// TIA Portal V17 export
// export: Created 2025-03-11T12:28:50.280284Z, ExportSetting WithDefaults, DisplayName Totally Integrated Automation Portal, DisplayVersion V17 Update 8, DisplayName TIA Portal Openness, DisplayVersion V17 Update 8, DisplayName TIA Portal Version Control Interface, DisplayVersion V17, DisplayName SINAMICS Startdrive Advanced, DisplayVersion V17 SP2, DisplayName SINAMICS Startdrive G110M, G120, G120C, G120D, G120P, G115D, DisplayVersion V17 SP2, DisplayName SINAMICS Startdrive G130, G150, S120, S150, SINAMICS MV, S210, DisplayVersion V17 SP2, DisplayName STEP 7 Professional, DisplayVersion V17 Update 8, DisplayName SINUMERIK ONE STEP 7 Toolbox, DisplayVersion V17 Update 12, DisplayName SINUMERIK 840D sl STEP 7 Toolbox, DisplayVersion V17 Update 12, DisplayName STEP 7 Safety, DisplayVersion V17 Update 6, DisplayName WinCC Advanced, DisplayVersion V17 Update 8
FUNCTION_BLOCK "FB21222_POWDER_FILLING_START_STOP_BY_CURRENT"   // FB21222, LAD
{ S7_Optimized_Access := 'TRUE' }
VERSION : 0.1
// stored: AutoNumber false, IsIECCheckEnabled false, IsRetainMemResEnabled false, MemoryReserve 100, SetENOAutomatically false, UDAEnableTagReadback false
   VAR_INPUT
      SENSOR_VALUE : Int;   // SENSOR VALUE
      iFEEDER_STATE_LINE : Word;
      HMI_HIGH_CURRENT_LIMIT : Real;   // HMI HIGH CURRENT LIMIT
      HMI_LOW_CURRENT_LIMIT : Real;   // HMI LOW CURRENT LIMIT
   END_VAR
   VAR_OUTPUT
      POWDER_FILLING_STOP_BY_CURRENT : Bool;   // HMI POWDER FILLING STOP BY CURRENT
      POWDER_FILLING_START_BY_CURRENT : Bool;   // HMI POWDER FILLING START BY CURRENT
   END_VAR
   VAR
      CURRENT_AVG_BLCK_START : Real;   // CURRENT AVERAGE BLOCK START
      CURRENT_AVG_BLCK_STOP : Real;   // CURRENT AVERAGE BLOCK STOP
      CURRENT_AVG_BLCK_HMI_START : Real;   // CURRENT AVERAGE BLOCK HMI START
      CURRENT_AVG_BLCK_HMI_STOP : Real;   // CURRENT AVERAGE BLOCK HMI STOP
      PF_LINE_ON : Bool;   // POWDER FEEDER LINE ON
      NORMALIZED_VALUE : Real;   // NORMALIZED
      SCALED_VALUE : Real;   // SCALED
      DB_CURRENT_AVERAGE_START : "FB21990_LGF_FloatingAverage";
      DB_CURRENT_AVERAGE_STOP { S7_SetPoint := 'True'} : "FB21990_LGF_FloatingAverage";
      TON_TIME { S7_SetPoint := 'True'} : TON_TIME;
   END_VAR
   VAR_TEMP   // added for the SCL form of the ladder/FBD networks
      _w1 : Bool;
   END_VAR
BEGIN

REGION Network 1: SCALE - CURRENT VALUE
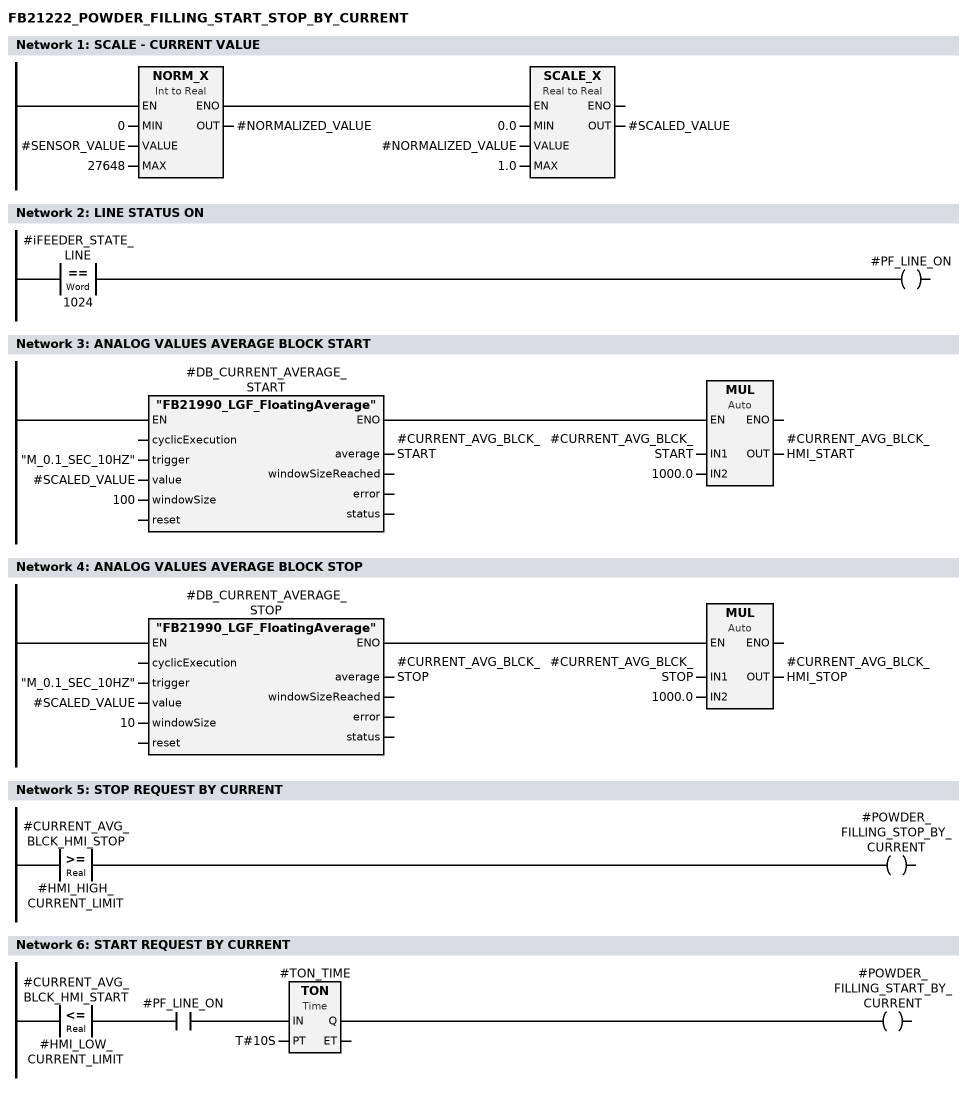
   RUNG wire#powerrail
      { S7_Templates := "[SrcType := Int, DestType := Real]"; S7_GenerateENO := "TRUE" } Normalize(min := 0, value := #SENSOR_VALUE, max := 27648, out => #NORMALIZED_VALUE)
      { S7_Templates := "[SrcType := Real, DestType := Real]"; S7_GenerateENO := "TRUE" } Scale(min := 0.0, value := #NORMALIZED_VALUE, max := 1.0, out => #SCALED_VALUE)
   END_RUNG
   // the same network as SCL:
   // ENO of a box is taken as its EN; it also drops when the box reports an error
   #NORMALIZED_VALUE := NORM_X(MIN := 0, VALUE := #SENSOR_VALUE, MAX := 27648);
   #SCALED_VALUE := SCALE_X(MIN := 0.0, VALUE := #NORMALIZED_VALUE, MAX := 1.0);
END_REGION

REGION Network 2: LINE STATUS ON
   RUNG wire#powerrail
      { S7_Templates := "SrcType := Word" } EQ_Contact(in1 := #iFEEDER_STATE_LINE, in2 := 1024)
      Coil( #PF_LINE_ON )
   END_RUNG
   // the same network as SCL:
   #PF_LINE_ON := #iFEEDER_STATE_LINE = 1024;
END_REGION

REGION Network 3: ANALOG VALUES AVERAGE BLOCK START
   RUNG wire#powerrail
      #DB_CURRENT_AVERAGE_START(cyclicExecution :=, trigger := "M_0.1_SEC_10HZ", value := #SCALED_VALUE, windowSize := 100, reset :=, average => #CURRENT_AVG_BLCK_START, windowSizeReached =>, error =>, status =>)
      { S7_GenerateENO := "TRUE" } Mul(in1 := #CURRENT_AVG_BLCK_START, in2 := 1000.0, out => #CURRENT_AVG_BLCK_HMI_START)
   END_RUNG
   // the same network as SCL:
   #DB_CURRENT_AVERAGE_START(trigger := "M_0.1_SEC_10HZ",   // "FB21990_LGF_FloatingAverage"
                           value := #SCALED_VALUE,
                           windowSize := 100,
                           average => #CURRENT_AVG_BLCK_START,
                           ENO => #_w1);
   IF #_w1 THEN #CURRENT_AVG_BLCK_HMI_START := #CURRENT_AVG_BLCK_START * 1000.0; END_IF;
END_REGION

REGION Network 4: ANALOG VALUES AVERAGE BLOCK STOP
   RUNG wire#powerrail
      #DB_CURRENT_AVERAGE_STOP(cyclicExecution :=, trigger := "M_0.1_SEC_10HZ", value := #SCALED_VALUE, windowSize := 10, reset :=, average => #CURRENT_AVG_BLCK_STOP, windowSizeReached =>, error =>, status =>)
      { S7_GenerateENO := "TRUE" } Mul(in1 := #CURRENT_AVG_BLCK_STOP, in2 := 1000.0, out => #CURRENT_AVG_BLCK_HMI_STOP)
   END_RUNG
   // the same network as SCL:
   #DB_CURRENT_AVERAGE_STOP(trigger := "M_0.1_SEC_10HZ",   // "FB21990_LGF_FloatingAverage"
                           value := #SCALED_VALUE,
                           windowSize := 10,
                           average => #CURRENT_AVG_BLCK_STOP,
                           ENO => #_w1);
   IF #_w1 THEN #CURRENT_AVG_BLCK_HMI_STOP := #CURRENT_AVG_BLCK_STOP * 1000.0; END_IF;
END_REGION

REGION Network 5: STOP REQUEST BY CURRENT
   RUNG wire#powerrail
      { S7_Templates := "SrcType := Real" } GE_Contact(in1 := #CURRENT_AVG_BLCK_HMI_STOP, in2 := #HMI_HIGH_CURRENT_LIMIT)
      Coil( #POWDER_FILLING_STOP_BY_CURRENT )
   END_RUNG
   // the same network as SCL:
   #POWDER_FILLING_STOP_BY_CURRENT := #CURRENT_AVG_BLCK_HMI_STOP >= #HMI_HIGH_CURRENT_LIMIT;
END_REGION

REGION Network 6: START REQUEST BY CURRENT
   RUNG wire#powerrail
      { S7_Templates := "SrcType := Real" } LE_Contact(in1 := #CURRENT_AVG_BLCK_HMI_START, in2 := #HMI_LOW_CURRENT_LIMIT)
      Contact( #PF_LINE_ON )
      { S7_Templates := "time_type := Time" } #TON_TIME.TON(pt := T#10S, et =>)
      Coil( #POWDER_FILLING_START_BY_CURRENT )
   END_RUNG
   // the same network as SCL:
   #TON_TIME(IN := (#CURRENT_AVG_BLCK_HMI_START <= #HMI_LOW_CURRENT_LIMIT) AND #PF_LINE_ON, PT := T#10S);   // TON
   #POWDER_FILLING_START_BY_CURRENT := #TON_TIME.Q;
END_REGION
END_FUNCTION_BLOCK
